//simple function use without insantiation
FUNCTION BuildString : I_StringBuilder
VAR_INPUT
	nSizeDest : UDINT;
END_VAR
VAR
END_VAR

IF nSizeDest = 0 THEN
	RETURN;
END_IF

//Create if nonExistend
IF GVL_Strings.pStringBuilder = 0 THEN
	GVL_Strings.pStringBuilder := __NEW(CStringbuilder);
END_IF

// TODO: zero interface return
IF GVL_Strings.pStringBuilder = 0 THEN
	ADSLOGSTR(msgCtrlMask:= ADSLOG_MSGTYPE_ERROR, msgFmtStr:='StringBuilder creation for GVL_Strings failed', '');
	RETURN;
END_IF

IF GVL_Strings.pPara = 0 THEN
	GVL_Strings.pPara := __NEW(ST_StringBuilderPara);
END_IF

// TODO: zero interface return
IF GVL_Strings.pPara = 0 THEN
	ADSLOGSTR(msgCtrlMask:= ADSLOG_MSGTYPE_ERROR, msgFmtStr:='ST_Para for GVL_Strings failed', '');
	RETURN;
END_IF

GVL_Strings.pPara^.MaxBufferSize := nSizeDest;

// adapt needed bufferSize
IF nSizeDest > GVL_Strings.pStringBuilder^.MaxBufferSize THEN
	GVL_Strings.pStringBuilder^.Reset(pPara:=GVL_Strings.pPara);
END_IF


BuildString := GVL_Strings.pStringBuilder^;

END_FUNCTION

(* stored: Version 1.1.0.1, ProductVersion 3.1.4024.13
   POU BuildString: Id {7fdda044-a55b-476d-bf32-bb4c822b6b15}, SpecialFunc None *)
